{attribute addProperty BoxType "EJ2522-0000-0022"}
{attribute addProperty Id "StatusAT %I*Status_30784993162"}
{attribute addProperty CRC "3116062718"}
{attribute addProperty SizeInBites "16"}
{attribute addProperty SizeInBytes "2"}
TYPE PTO_Status_Channel_B9BB57FE :
STRUCT
	{attribute addProperty Name "Status"}
	Status AT %I* : Status_30784993;
END_STRUCT
END_TYPE

(* stored: Version 1.2.0.0, ProductVersion 3.1.4024.9
   DUT PTO_Status_Channel_B9BB57FE: Id {3ae66a90-7f21-4f5c-9e27-e3b2b589f886} *)
